PROGRAM MAIN
VAR

END_VAR

END_PROGRAM

(* stored: Version 1.1.0.1, ProductVersion 3.1.4024.13
   POU MAIN: Id {352c01da-1586-42c5-b1d3-30a80a0c5354}, SpecialFunc None *)
